FUNCTION derivcvar_M_p_t3: REAL
{ S7_Optimized_Access := 'false' }
    VAR_INPUT
        state: STATE;
    END_VAR

BEGIN
    derivcvar_M_p_t3 := state.cvar_M_p_t3;
END_FUNCTION
